# B&R Automation Studio project EnergyMon
Automation Studio 4.4.6.71 SP

## Configuration Config1

CPU , AutomationRuntime C2.31, Build 2.95.3, Vc V3.73.4

### Hardware
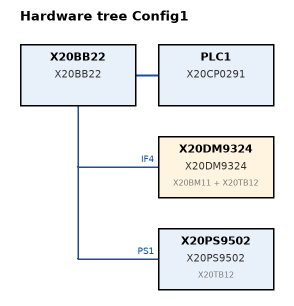
```
PLC1 : X20CP0291 v1.0.3.0  [SL -> X20BB22.SL1]
  Connector IF2:
    Mode = DHCP Client
    InternetAddress = 192.168.0.1
    SubnetMask = 255.255.0.0
  AnalogPermanentMemory = 128
  DigitalPermanentMemory = 128
  BRObjects = 150
  RebootReset = 2
  RebootPowerfail = 2
  Connections = 3
  PVTables = 0
  DelayPowerFail = 0
  NrOfExceptionObjects = 0
  ExceptionUserStack = 8
  ExceptionIrqStack = 896
  CyclicTaskClassCount = 2
X20BB22 : X20BB22 v1.0.2.0
X20BM11 : X20BM11 v1.0.0.1  [X2X1 -> X20BB22.IF4]
X20DM9324 : X20DM9324 v1.0.4.0  [SS1 -> X20TB12a.SS; SL -> X20BM11.SL1]
X20PS9502 : X20PS9502 v1.0.0.0  [PS -> X20BB22.PS1; SS1 -> X20TB12.SS]
X20TB12 : X20TB12 v1.0.0.0
X20TB12a : X20TB12 v1.0.0.0
```

### Cpu.per - PLC1/Cpu.per
```iecst
(********************************************************************
 * COPYRIGHT --
 ********************************************************************
 * File: Cpu.per
 * Author: Petr Fišer
 * Created: June 19, 2013
 ********************************************************************
 * Declaration of permanent variables
 ********************************************************************)
VAR_CONFIG
	gInitDone AT %MX0;
	gTrigger1Value AT %MW0;
	gTrigger1DeadTime AT %MD2;
	gTrigger2Value AT %MW6;
	gTrigger2DeadTime AT %MD8;
END_VAR
```

### IoMap.iom - PLC1/IoMap.iom
```iecst
(********************************************************************
 * COPYRIGHT --
 ********************************************************************
 * File: IoMap.iom
 * Author: Petr Fišer
 * Created: June 19, 2013
 ********************************************************************
 * IO mapping file
 ********************************************************************)
VAR_CONFIG
	::Main:realPowerProcess.diS0 AT %IX."X20DM9324".DigitalInput01;
	::Main:reactivePowerProcess.diS0 AT %IX."X20DM9324".DigitalInput02;
	::Main:diTarif AT %IX."X20DM9324".DigitalInput04;
	::Main:doTrigger1Sound AT %QX."X20DM9324".DigitalOutput01;
	::Main:doTrigger2Sound AT %QX."X20DM9324".DigitalOutput02;
	::Main:diAlarm1Reset AT %IX."X20DM9324".DigitalInput05;
	::Main:diAlarm2Reset AT %IX."X20DM9324".DigitalInput06;
	::Main:doTrigger1Light AT %QX."X20DM9324".DigitalOutput03;
	::Main:doTrigger2Light AT %QX."X20DM9324".DigitalOutput04;
END_VAR
```

## Logical view

Binary libraries used (declarations not repeated): Convert, runtime, operator, brsystem, astime

### Global.var - Global variables
```iecst
VAR RETAIN
	gInitDone : BOOL;
	gPowerFactor : REAL;
	gPowerLimit : REAL;
	gTarifInterval : INT;
	gTrigger1Value : INT;
	gTrigger2Value : INT;
	gTrigger1DeadTime : DINT;
	gTrigger2DeadTime : DINT;
END_VAR
VAR
	gTrigger1MuteActive : BOOL;
	gTrigger2MuteActive : BOOL;
	gTrigger1Alarm : BOOL;
	gTrigger2Alarm : BOOL;
	gActPower : REAL;
	gPeakPower : REAL;
	gPowerConsumed : REAL;
	gPowerLimitInterval : REAL;
	gTarifTime : DATE_AND_TIME;
END_VAR
```


### Program Logical/Main (ANSIC)

#### Main.c - Implementation code
```c
/********************************************************************
 * COPYRIGHT --
 ********************************************************************
 * Program: Main
 * File: Main.c
 * Author: Petr Fišer
 * Created: June 01, 2013
 ********************************************************************
 * Implementation of program Main
 ********************************************************************/

#include <bur/plctypes.h>

#ifdef _DEFAULT_INCLUDES
	#include <AsDefault.h>
#endif

void _INIT MainInit(void)
{
    fbRTInfo.enable = 1;
    RTInfo(&fbRTInfo);
    cycleTime = fbRTInfo.cycle_time / 1000;

	if (!gInitDone)
	{
		gInitDone = 1;
		gPowerFactor = 0.1;
		gTarifInterval = 15;
		gPowerLimit = 160; // kWh
		gTrigger1Value = 100; // kWh
		gTrigger1DeadTime = 60 * 1000; // 1min.
		gTrigger2Value = 100; // kWh
		gTrigger2DeadTime = 30 * 1000; // 1min.
	}
}

void _CYCLIC MainCyclic(void)
{
	tarifFactor = 60.0 / gTarifInterval;
	gPowerLimitInterval = gPowerLimit / tarifFactor;

    //
    // Vypocet realneho vykonu ------------------------------------------------
    //
    //
    //

	realPowerProcess.factor = gPowerFactor; // kWh/imp.
    realPowerProcess.impPerHour = 1 / realPowerProcess.factor;

    realPowerProcess.actualTime += cycleTime;

    if (realPowerProcess.diS0)
    {
        if (!realPowerProcess.trigS0)
        {
            realPowerProcess.trigS0 = 1;
    	    realPowerProcess.period = realPowerProcess.actualTime;
            realPowerProcess.sumPower += realPowerProcess.factor;
            realPowerProcess.impCount++;
            realPowerProcess.actualTime = 0;
        }
    }
    else
        realPowerProcess.trigS0 = 0;

    tmpPeriod = realPowerProcess.actualTime;
    if (tmpPeriod < realPowerProcess.period)
        tmpPeriod = realPowerProcess.period;
    if (tmpPeriod > 0.0 && realPowerProcess.factor > 0.0)
        realPowerProcess.actPower = 3600000 / (tmpPeriod * realPowerProcess.impPerHour);
    if (realPowerProcess.actPower > realPowerProcess.peak)
        realPowerProcess.peak = realPowerProcess.actPower;

    //
    // Vypocet jaloveho vykonu ------------------------------------------------
    //
    //
    //

	reactivePowerProcess.factor = gPowerFactor; // kWh/imp.
    reactivePowerProcess.impPerHour = 1 / reactivePowerProcess.factor;

    reactivePowerProcess.actualTime += cycleTime;

    if (reactivePowerProcess.diS0)
    {
        if (!reactivePowerProcess.trigS0)
        {
            reactivePowerProcess.trigS0 = 1;
            reactivePowerProcess.period = reactivePowerProcess.actualTime;
            reactivePowerProcess.sumPower += reactivePowerProcess.factor;
            reactivePowerProcess.impCount++;
            reactivePowerProcess.actualTime = 0;
        }
    }
    else
        reactivePowerProcess.trigS0 = 0;

    tmpPeriod = reactivePowerProcess.actualTime;
    if (tmpPeriod < reactivePowerProcess.period)
        tmpPeriod = reactivePowerProcess.period;
    if (tmpPeriod > 0.0 && reactivePowerProcess.factor > 0.0)
        reactivePowerProcess.actPower = 3600000 / (tmpPeriod * reactivePowerProcess.impPerHour);
    if (reactivePowerProcess.actPower > reactivePowerProcess.peak)
        reactivePowerProcess.peak = reactivePowerProcess.actPower;

    //
    // Tarifni impuls ---------------------------------------------------------
    //
    //
    //

    if (!diTarif)
    {
        if (!trigTarif)
        {
            trigTarif = 1;

            fbGetTime.enable = 1;
            DTGetTime(&fbGetTime);
            if (!fbGetTime.status)
            {
				gTarifTime = fbGetTime.DT1;

				// Uloz data do statistiky.
				if (historyListNextItemIndex > MAX_HISTORY_LIST)
					historyListNextItemIndex = 0;

                historyList[historyListNextItemIndex].DateTime = fbGetTime.DT1;
                historyList[historyListNextItemIndex].sumRealPower = realPowerProcess.sumPower * tarifFactor;
                historyList[historyListNextItemIndex].sumReactivePower = reactivePowerProcess.sumPower * tarifFactor;
                historyList[historyListNextItemIndex].realMax = realPowerProcess.peak;
                historyList[historyListNextItemIndex].reactiveMax = reactivePowerProcess.peak;

                historyListNextItemIndex++;
            }

            realPowerProcess.sumPower = 0;
            realPowerProcess.peak = 0;
            reactivePowerProcess.sumPower = 0;
            reactivePowerProcess.peak = 0;
        }
    }
    else
        trigTarif = 0;

    //
    // Reset mereni a historie ------------------------------------------------
    //
    //
    //

    if (reset)
    {
        reset = 0;
        realPowerProcess.impCount = 0;
        realPowerProcess.period = 0;
        realPowerProcess.sumPower = 0;

        reactivePowerProcess.impCount = 0;
        reactivePowerProcess.period = 0;
        reactivePowerProcess.sumPower = 0;

        memset(&historyList, 0, sizeof(historyList));
        historyListNextItemIndex = 0;
    }

    //
    // Hlidej hodnotu max. vykonu ---------------------------------------------
    //
    //
    //

    gActPower = realPowerProcess.actPower + reactivePowerProcess.actPower;
    gPeakPower = realPowerProcess.peak + reactivePowerProcess.peak;
	gPowerConsumed = realPowerProcess.sumPower + reactivePowerProcess.sumPower;

	// Hlidani 1 -----------------------------------------------------------------
    if (gActPower > gTrigger1Value)
    {
		if (trigger1Delay > 0)
			trigger1Delay -= cycleTime;
		else
			gTrigger1Alarm = 1;
    }
	else
	{
		trigger1Delay = (gTrigger1DeadTime * 1000);
		gTrigger1MuteActive = 0;
		gTrigger1Alarm = 0;
	}

	// Rucni potvrzeni alarmu tlacitkem.
	if (diAlarm1Reset)
		gTrigger1MuteActive = 1;

	doTrigger1Sound = !gTrigger1MuteActive && gTrigger1Alarm;
	doTrigger1Light = gTrigger1Alarm;

	// Hlidani 2 -----------------------------------------------------------------
	if (gActPower > gTrigger2Value)
	{
		if (trigger2Delay > 0)
			trigger2Delay -= cycleTime;
		else
			gTrigger2Alarm = 1;
	}
	else
	{
		trigger2Delay = (gTrigger2DeadTime * 1000);
		gTrigger2MuteActive = 0;
		gTrigger2Alarm = 0;
	}

	// Rucni potvrzeni alarmu tlacitkem.
	if (diAlarm2Reset)
		gTrigger2MuteActive = 1;

	doTrigger2Sound = !gTrigger2MuteActive && gTrigger2Alarm;
	doTrigger2Light = gTrigger2Alarm;
}
```

#### Main.typ - Local data types
```iecst
TYPE
	MeasurementProcess_typ : 	STRUCT
		diS0 : BOOL;
		actualTime : TIME;
		period : TIME;
		factor : REAL;
		sumPower : REAL;
		actPower : REAL;
		trigS0 : BOOL;
		impCount : UDINT;
		impPerHour : REAL;
		peak : REAL;
	END_STRUCT;
	HistoryItem_typ : 	STRUCT
		DateTime : DATE_AND_TIME;
		sumRealPower : REAL;
		sumReactivePower : REAL;
		realMax : REAL;
		reactiveMax : REAL;
	END_STRUCT;
END_TYPE
```

#### Main.var - Local variables
```iecst
VAR CONSTANT
	MAX_HISTORY_LIST : UINT := 95;
END_VAR
VAR
	realPowerProcess : MeasurementProcess_typ;
	reactivePowerProcess : MeasurementProcess_typ;
	tmpPeriod : TIME;
	fbRTInfo : RTInfo := (0);
	cycleTime : REAL;
END_VAR
VAR RETAIN
	historyList : ARRAY[0..MAX_HISTORY_LIST] OF HistoryItem_typ;
	historyListNextItemIndex : UINT;
END_VAR
VAR
	fbGetTime : DTGetTime;
	reset : BOOL;
	diTarif : BOOL;
	diAlarm1Reset : BOOL;
	diAlarm2Reset : BOOL;
	trigTarif : BOOL;
	tarifFactor : REAL;
	doTrigger1Sound : BOOL;
	doTrigger2Sound : BOOL;
	doTrigger1Light : BOOL;
	doTrigger2Light : BOOL;
	trigger1Delay : DINT;
	trigger2Delay : DINT;
END_VAR
```

### Program Logical/Test (ANSIC) - A new program

#### Test.c - Implementation code
```c
/********************************************************************
 * COPYRIGHT --
 ********************************************************************
 * Program: Test
 * File: Test.c
 * Author: Petr Fišer
 * Created: June 23, 2013
 ********************************************************************
 * Implementation of program Test
 ********************************************************************/

#include <bur/plctypes.h>

#ifdef _DEFAULT_INCLUDES
 #include <AsDefault.h>
#endif

void _INIT TestINIT( void )
{
	pulsePeriod = 10 * 1000; // 10 sek.
    tarifPeriod = 15 * 60 * 1000; // 15 min.
}

void _CYCLIC TestCYCLIC( void )
{
    doPulse = 0;
    doTarif = 0;

	timer += 10;
    if (timer >= pulsePeriod)
    {
        timer = 0;
        pulseDelay = 500;
    }

    if (pulseDelay > 0)
    {
        pulseDelay -= 10;
        doPulse = 1;
    }

    tarifTimer += 10;
    if (tarifTimer >= tarifPeriod)
    {
        tarifTimer = 0;
        tarifDelay = 500;
    }

    if (tarifDelay > 0)
    {
        tarifDelay -= 10;
        doTarif = 1;
    }
}
```

#### Test.var - Local variables
```iecst
VAR
	timer : UDINT;
	doPulse : BOOL;
	doTarif : BOOL;
	pulseDelay : INT;
	pulsePeriod : UDINT;
	tarifDelay : INT;
	tarifPeriod : UDINT;
	tarifTimer : UDINT;
END_VAR
```

Listed in the project but not available here: Logical/Global.typ
